(* PLC project TrafficLight, AutonomyLogic OpenPLC Editor 3.0 *)
(* stored: creationDateTime 2026-01-15T10:00:00, version 1.0, modificationDateTime 2026-07-24T08:00:00 *)

TYPE TRAFFIC_STATE : DINT := 0;
END_TYPE

TYPE DIAGNOSTIC_STRUCT : STRUCT
  errorCode : INT;
  severity : USINT;
  timestamp : TIME;
END_STRUCT;
END_TYPE

FUNCTION_BLOCK TrafficTimer
  VAR_INPUT
    preset : TIME := T#5s;
    enable : BOOL;
  END_VAR
  VAR_OUTPUT
    elapsed : TIME;
    done : BOOL;
  END_VAR
  VAR
    ton1 : TON;
    accumulator : DINT;
  END_VAR

            
(* Traffic timer with edge-triggered enable *)
ton1(IN := enable, PT := preset);

IF NOT enable THEN
  elapsed := T#0s;
  done := FALSE;
  accumulator := 0;
END_IF;

IF ton1.Q THEN
  elapsed := ton1.ET;
  done := TRUE;
  accumulator := accumulator + 1;
END_IF;

          
END_FUNCTION_BLOCK

FUNCTION NextState : INT
  VAR_INPUT
    current : TRAFFIC_STATE;
    overrideReq : BOOL;
  END_VAR

            
// Emergency override has highest priority
IF overrideReq THEN
  NextState := 0;  (* FLASHING_RED *)
  RETURN;
END_IF;

// Normal state machine
CASE current OF
  0:  // RED → GREEN after delay
    NextState := 1;
  1:  // GREEN → YELLOW after delay
    NextState := 2;
  2:  // YELLOW → RED after delay
    NextState := 0;
  3:  // FLASHING mode
    NextState := 4;
  4:
    NextState := 3;
END_CASE;

          
END_FUNCTION

PROGRAM main
  VAR
    state : TRAFFIC_STATE := 0;
    redLight : BOOL;
    yellowLight : BOOL;
    greenLight : BOOL;
    phaseTimer : TrafficTimer;
    emergencyStop : BOOL;
    loopCounter : DINT;
  END_VAR
  VAR_INPUT
    systemClock : TIME;
  END_VAR
  VAR_OUTPUT
    statusWord : INT;
  END_VAR
  VAR_IN_OUT
    configBlock : DIAGNOSTIC_STRUCT;
  END_VAR
  VAR_TEMP
    tmpResult : DINT;
  END_VAR

            
(* Main traffic light controller *)
state := NextState(state, emergencyStop);

(* Configure timer based on state *)
CASE state OF
  0:  // RED phase
    redLight := TRUE;
    yellowLight := FALSE;
    greenLight := FALSE;
    phaseTimer.enable := FALSE;
    phaseTimer.preset := T#30s;

  1:  // GREEN phase
    redLight := FALSE;
    greenLight := TRUE;
    phaseTimer.enable := TRUE;
    phaseTimer.preset := T#30s;

  2:  // YELLOW phase
    greenLight := FALSE;
    yellowLight := TRUE;
    phaseTimer.enable := TRUE;
    phaseTimer.preset := T#5s;

  3:  // FLASHING_RED (emergency)
    ldToggle := NOT ldToggle;
    redLight := ldToggle;
    yellowLight := FALSE;
    greenLight := FALSE;
    statusWord := statusWord + 1;
END_CASE;

(* Update timer *)
phaseTimer();

(* Loop counting *)
FOR loopCounter := 0 TO 1000 DO
  tmpResult := loopCounter * 2;
  IF tmpResult > 500 THEN
    EXIT;
  END_IF;
END_FOR;

          
END_PROGRAM

FUNCTION_BLOCK DiagnosticLogger
  VAR
    logIndex : DINT;
    logArray : ARRAY[0..99] OF STRING;
  END_VAR

            
WHILE logIndex < 100 DO
  logArray[logIndex] := '';
  logIndex := logIndex + 1;
END_WHILE;

          
END_FUNCTION_BLOCK

FUNCTION_BLOCK R_TRIG_Impl
  VAR_INPUT
    CLK : BOOL;
  END_VAR
  VAR_OUTPUT
    Q : BOOL;
  END_VAR
  VAR
    M : BOOL := FALSE;
  END_VAR

            
Q := CLK AND NOT M;
M := CLK;

          
END_FUNCTION_BLOCK

CONFIGURATION DefaultConfig
  RESOURCE RaspberryPi ON PLC
    TASK FastTask(INTERVAL := 20ms, PRIORITY := 10);
    TASK SlowTask(INTERVAL := 100ms, PRIORITY := 20);
    PROGRAM mainInstance WITH FastTask : main;
    PROGRAM diagInstance WITH SlowTask : DiagnosticLogger;
  END_RESOURCE
END_CONFIGURATION
